{attribute 'linkalways'}
{attribute 'no_explicit_call' := 'do not call this POU directly'}
FUNCTION_BLOCK TaskCyclicEvent EXTENDS Event IMPLEMENTS I_TaskCyclicEvent
VAR
	parent : I_Task;
END_VAR

METHOD FB_init : BOOL
VAR_INPUT
	bInitRetains : BOOL; // if TRUE, the retain variables are initialized (warm start / cold start)
	bInCopyCode : BOOL;  // if TRUE, the instance afterwards gets moved into the copy code (online change)
	Parent : I_Task;
END_VAR
this^.parent := Parent;
END_METHOD

PROPERTY Info : PlcTaskSystemInfo
GET
Info := parent.Info;
END_GET
END_PROPERTY

METHOD PUBLIC Notify
VAR_INPUT
END_VAR
NotifySubscribers();
END_METHOD

END_FUNCTION_BLOCK

(* stored: Version 1.1.0.1, ProductVersion 3.1.4024.11
   POU TaskCyclicEvent: Id {f887109a-3ad6-453d-bf0f-4c5420be9500}, SpecialFunc None
   Method FB_init: Id {34690361-5385-45c4-abe3-fc0b1ad447c4}
   Property Info: Id {45316dd5-4217-4539-8f58-db0230a3c479}
   Get Get: Id {68fc8d6f-9547-47bb-b1df-12254bd63a37}
   Method Notify: Id {7ce2d076-8003-40b7-b652-f32bcd386fbe} *)
